FUNCTION_BLOCK FB_TankControl (* Basic Function Block Type *)
  (* Standard: 61499-2 *)
  (* Version 0.0, 2014-5-4, wildai, nxtControl GmbH, Template *)
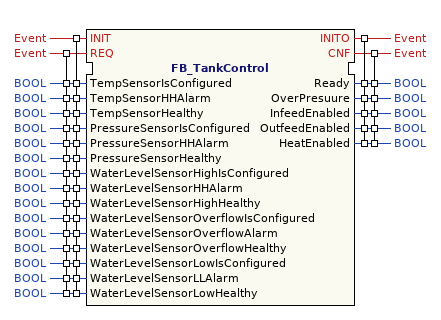
  EVENT_INPUT
    INIT WITH TempSensorIsConfigured, TempSensorHHAlarm, TempSensorHealthy, PressureSensorIsConfigured, PressureSensorHHAlarm, PressureSensorHealthy, WaterLevelSensorHighIsConfigured, WaterLevelSensorHHAlarm, WaterLevelSensorHighHealthy, WaterLevelSensorOverflowIsConfigured, WaterLevelSensorOverflowAlarm, WaterLevelSensorOverflowHealthy, WaterLevelSensorLowIsConfigured, WaterLevelSensorLLAlarm, WaterLevelSensorLowHealthy; (* Initialization Request *)
    REQ WITH TempSensorIsConfigured, TempSensorHHAlarm, TempSensorHealthy, PressureSensorIsConfigured, PressureSensorHHAlarm, PressureSensorHealthy, WaterLevelSensorHighIsConfigured, WaterLevelSensorHHAlarm, WaterLevelSensorHighHealthy, WaterLevelSensorOverflowIsConfigured, WaterLevelSensorOverflowAlarm, WaterLevelSensorOverflowHealthy, WaterLevelSensorLowIsConfigured, WaterLevelSensorLLAlarm, WaterLevelSensorLowHealthy; (* Normal Execution Request *)
  END_EVENT
  EVENT_OUTPUT
    INITO WITH Ready, OverPresuure, InfeedEnabled, OutfeedEnabled, HeatEnabled; (* Initialization Confirm *)
    CNF WITH Ready, OverPresuure, InfeedEnabled, OutfeedEnabled, HeatEnabled; (* Execution Confirmation *)
  END_EVENT
  VAR_INPUT
    TempSensorIsConfigured : BOOL;
    TempSensorHHAlarm : BOOL;
    TempSensorHealthy : BOOL;
    PressureSensorIsConfigured : BOOL;
    PressureSensorHHAlarm : BOOL;
    PressureSensorHealthy : BOOL;
    WaterLevelSensorHighIsConfigured : BOOL;
    WaterLevelSensorHHAlarm : BOOL;
    WaterLevelSensorHighHealthy : BOOL;
    WaterLevelSensorOverflowIsConfigured : BOOL;
    WaterLevelSensorOverflowAlarm : BOOL;
    WaterLevelSensorOverflowHealthy : BOOL;
    WaterLevelSensorLowIsConfigured : BOOL;
    WaterLevelSensorLLAlarm : BOOL;
    WaterLevelSensorLowHealthy : BOOL;
  END_VAR
  VAR_OUTPUT
    Ready : BOOL;
    OverPresuure : BOOL;
    InfeedEnabled : BOOL;
    OutfeedEnabled : BOOL;
    HeatEnabled : BOOL;
  END_VAR
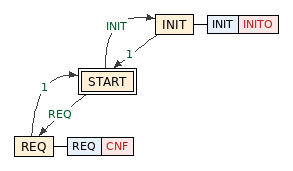
  EC_STATES
    START; (* Initial State *)
    INIT : INIT -> INITO; (* Initialization *)
    REQ : REQ -> CNF; (* Normal execution *)
  END_STATES
  EC_TRANSITIONS
    START TO INIT := INIT;
    INIT TO START := 1;
    START TO REQ := REQ;
    REQ TO START := 1;
  END_TRANSITIONS
  ALGORITHM INIT IN ST: (* Initialization algorithm *)
;
Ready := FALSE;
OverPresuure := FALSE;
InfeedEnabled := FALSE;
OutfeedEnabled := FALSE;
HeatEnabled := FALSE;
  END_ALGORITHM
  ALGORITHM REQ IN ST: (* Normally executed algorithm *)
;

IF ((TempSensorIsConfigured AND NOT TempSensorHealthy) OR
	(PressureSensorIsConfigured AND NOT PressureSensorHealthy) OR
	(WaterLevelSensorHighIsConfigured AND NOT WaterLevelSensorHighHealthy) OR
	(WaterLevelSensorOverflowIsConfigured AND NOT WaterLevelSensorOverflowHealthy) OR
	(WaterLevelSensorLowIsConfigured AND NOT WaterLevelSensorLowHealthy)) THEN
	Ready := FALSE;
ELSE
	Ready := TRUE;
END_IF;

IF ((TempSensorIsConfigured AND NOT TempSensorHHAlarm) AND Ready) THEN
	HeatEnabled := TRUE;
ELSE
	HeatEnabled := FALSE;
END_IF;

IF (PressureSensorIsConfigured AND PressureSensorHHAlarm) THEN
	OverPresuure := TRUE;
ELSE
	OverPresuure := FALSE;
END_IF;

IF ((WaterLevelSensorHighIsConfigured AND WaterLevelSensorHHAlarm) OR (WaterLevelSensorOverflowIsConfigured AND WaterLevelSensorOverflowAlarm) OR NOT Ready OR (NOT WaterLevelSensorHighIsConfigured AND NOT WaterLevelSensorOverflowIsConfigured)) THEN
	InfeedEnabled := FALSE;
ELSE
	InfeedEnabled := TRUE;
END_IF;

IF ((WaterLevelSensorLowIsConfigured AND NOT WaterLevelSensorLLAlarm) AND Ready) THEN
	OutfeedEnabled := TRUE;
ELSE
	OutfeedEnabled := FALSE;
END_IF;
  END_ALGORITHM
END_FUNCTION_BLOCK
